FUNCTION_BLOCK DumpStation
VAR_INPUT
END_VAR
VAR_OUTPUT
END_VAR
VAR
END_VAR

// NETWORK 1

END_FUNCTION_BLOCK

(* stored: Version 1.1.0.1, ProductVersion 3.1.0.25
   POU DumpStation: Id {08442602-941f-4bfa-8c69-7c3689b50361} *)
